// SIMATIC S7-200 project (STEP 7-Micro/WIN), CPU 226 REL 02.00

ORGANIZATION_BLOCK MAIN:OB1
TITLE=PROGRAM COMMENTS
BEGIN
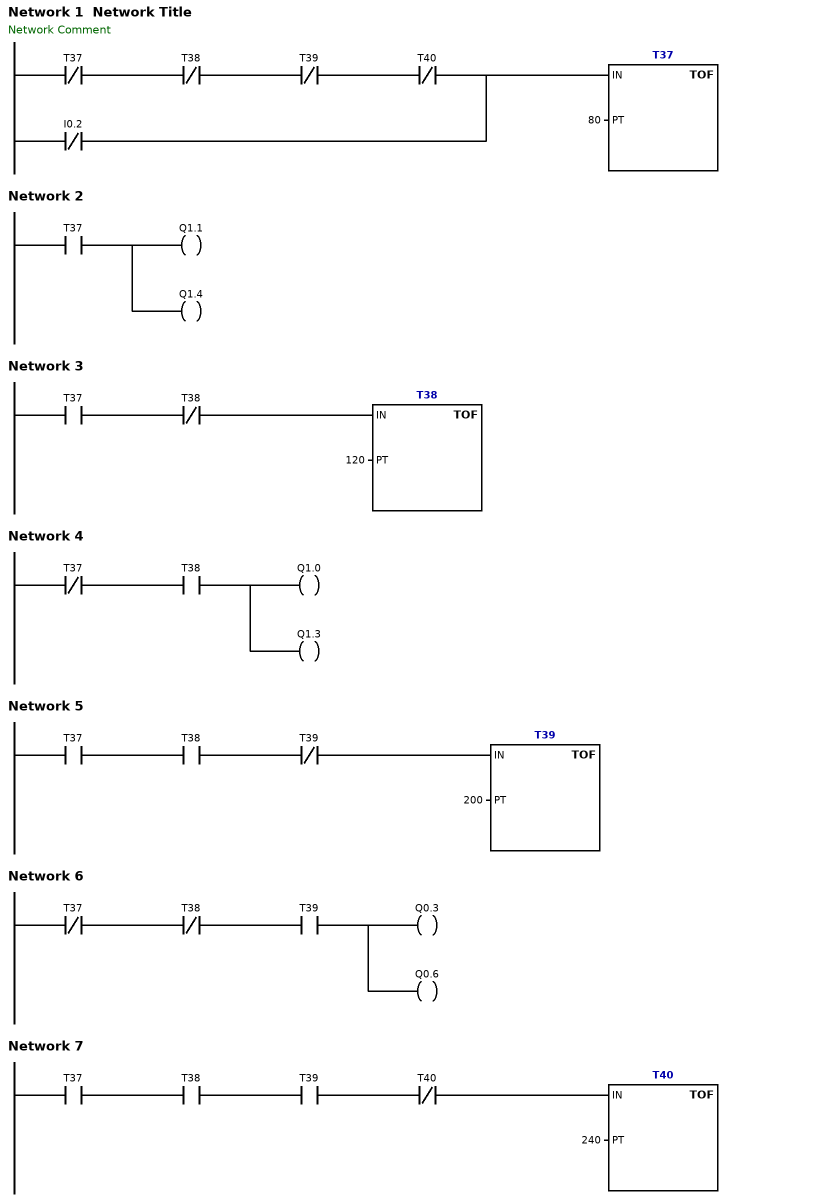
Network 1 // Network Title
// Network Comment
// (network saved uncompiled; LAD cells follow)
// row 0: c0 -|/|- T37  c1 -|/|- T38  c2 -|/|- T39  c3 -|/|- T40 v  c4 --  c5 [TOF T37 IN:=power@row0, PT:=80]
// row 1: c0 -|/|- I0.2  c1 --  c2 --  c3 -- ^  c5 [box]
Network 2
LD     T37
=      Q1.1
=      Q1.4
Network 3
LD     T37
AN     T38
TOF    T38, 120
Network 4
LDN    T37
A      T38
=      Q1.0
=      Q1.3
Network 5
LD     T37
A      T38
AN     T39
TOF    T39, 200
Network 6
LDN    T37
AN     T38
A      T39
=      Q0.3
=      Q0.6
Network 7
LD     T37
A      T38
A      T39
AN     T40
TOF    T40, 240
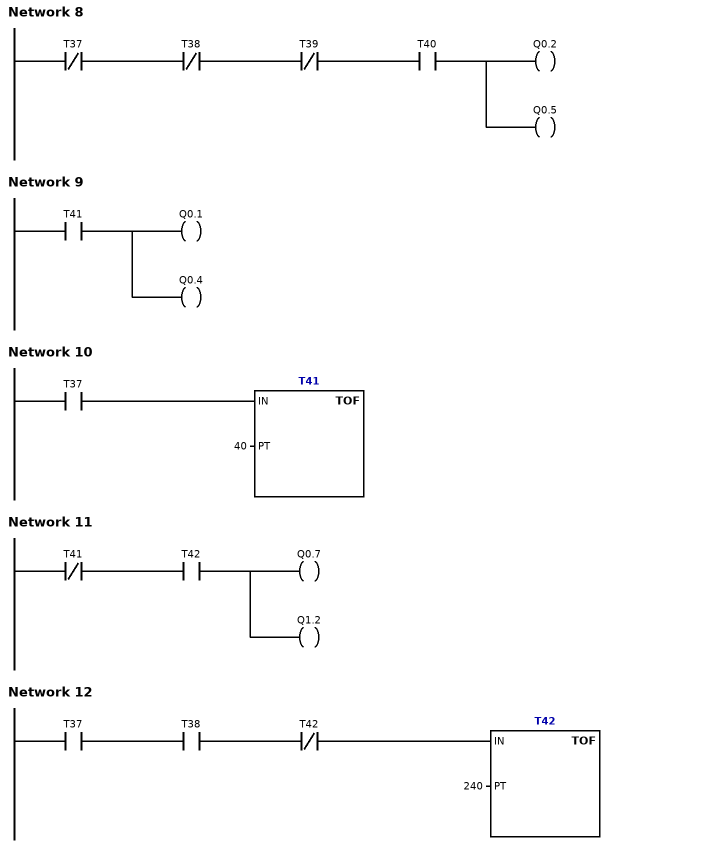
Network 8
LDN    T37
AN     T38
AN     T39
A      T40
=      Q0.2
=      Q0.5
Network 9
LD     T41
=      Q0.1
=      Q0.4
Network 10
LD     T37
TOF    T41, 40
Network 11
LDN    T41
A      T42
=      Q0.7
=      Q1.2
Network 12
LD     T37
A      T38
AN     T42
TOF    T42, 240
END_ORGANIZATION_BLOCK
